# EPICS autosave request: exampleApp/Db/ADCSimDetector_settings.req
$(P)$(R)TimeStep
$(P)$(R)NumTimePoints

file "NDArrayBase_settings.req", P=$(P), R=$(R)
